Universal Robots PolyScope program: comunicacio2.urp

Program comunicacio2 (installation=default directory=/programs createdIn=5.9.3.1031212 lastSavedIn=5.9.3.1031212 robotSerialNumber=20195300809)
Calibrated DH parameters: a=[-0.000085, -0.20076, -0.212369, 0.000121, -0.000118, 0]; d=[0.15185, -26.306375, 24.753047, 1.684739, 0.085386, 0.092088]; alpha=[1.572149, -0.00522, -0.011864, 1.571339, -1.571085, 0]; deltaTheta=[0, 0.599885, -0.513355, -0.086555, 0.000006, 0]
BeforeStart
  var_1 := socket_open("10.5.20.84",30001)
  Loop_1 := False
Robot Program (runOnlyOnce=false)
  Loop Counting (count=4) loopVariable(name=Loop_2)
    Loop_1 := socket_open("10.5.20.90",30001)
    Wait Sleep waitTime=0.5
    str := "Missatge enviat"
    Script: socket_send_string(str)
    Script: msg=socket_read_string(timeout=3)
    If msg≟"Missatge rebut"
      str := "Digues hola o adeu"
    If msg≠"No s'ha rebut missatge: Error de comunicacio"
      Script: socket_send_string("No s'ha rebut missatge")
      Script: socket_close()
    Script: socket_send_string(str)
    Script: msg=socket_read_string(timeout=3)
    If msg≟"hola"
      Script: socket_send_string("Me has saludado")
    If msg≟"adeu"
      Script: socket_send_string("Te has despedido")
    Script: socket_close()
